TEXTLIST txlCompresorTypes
  1 = '8P0'
  2 = 'Volvo CMA'
   = ''
END_TEXTLIST

(* stored: Version 1.1.0.1, ProductVersion 3.1.4024.12
   TextList txlCompresorTypes: Id {e445201f-2382-4c0b-a8a6-6b8317a23f40} *)
